TYPE U_OdriveSetInputVelBytes :
UNION
    stSetInputVel : ST_OdriveSetInputVel;
    aBytes : ARRAY[0..7] OF BYTE;
END_UNION
END_TYPE

(* stored: Version 1.1.0.1
   DUT U_OdriveSetInputVelBytes: Id {2c726f47-1d6b-4712-8b2c-429307443024} *)
